PROGRAM MAIN
VAR
END_VAR

END_PROGRAM

(* stored: Version 1.1.0.1, ProductVersion 3.1.4020.12
   POU MAIN: Id {9c1ccd94-44ac-4d01-9618-7d667ac8f86e}, SpecialFunc None *)
